// TIA Portal V18 export
TYPE "UDT_HSsDI"
// stored: IsFailsafeCompliant false
   STRUCT
      xBoilerShuntPumpReady : Array[1..2] of Bool;
      xBoilerShuntPumpInd : Array[1..2] of Bool;
      xBoilerShuntPumpAlarm : Array[1..2] of Bool;
      xBoilerShuntPumpInAuto : Array[1..2] of Bool;
      xBoilerStage1Ind : Array[1..2] of Bool;
      xBoilerStage2Ind : Array[1..2] of Bool;
      xBurnerAlarm : Array[1..2] of Bool;
      xBoilerAlarm : Array[1..2] of Bool;
      xBoilerReady : Array[1..2] of Bool;
      xBoilerReserve : Array[1..2] of Bool;
      xSeasonWinter : Array[1..2] of Bool;
      xSeasonSummer : Array[1..2] of Bool;
      xSeasonAuto : Array[1..2] of Bool;
      xBoilerWaterLvl : Array[1..2] of Bool;
      xBoilerPmin : Array[1..2] of Bool;
      xBoilerPmax : Array[1..2] of Bool;
   END_STRUCT;
   // xBoilerShuntPumpReady[1..2] := true;
END_TYPE
